//----------------------------------------------------------------------------//
//            Copyright 2018 Rieckermann Engineering Operations               //
//                Automatically Generated File - Do Not Edit                  //
//----------------------------------------------------------------------------//
// Description:                                                               //
// This file contains globally addressable event words for process alarms and //
// messages to be logged.                                                     //
//----------------------------------------------------------------------------//
// Revision history:                                                          //
// Rev By               Date        CC        Note                            //
// 1.1 David Paspa      10-Aug-2018 NA        Convert triggers to word bits.  //
// 1.0 David Paspa      14-May-2018 NA        Initial design for S7-1500.     //
//----------------------------------------------------------------------------//
DATA_BLOCK "dbEVENT"
TITLE = Global messages bits
{ S7_Optimized_Access := 'TRUE' }
AUTHOR : REO
NAME : dbEVENT
VERSION : 1.1

STRUCT
    alarmBlock : STRUCT                          // Block related alarms
@@TEMPLATE_BEGIN|createLevelsGlobal@@
@@ATTR_BEGIN|createClassesForLevel@@
@@ATTR_BEGIN|createInstancesGlobal@@
        alarm_@@INSTANCE@@ : Int;                // @@CLASS@@ block alarms
@@ATTR_END|createInstancesGlobal@@
@@ATTR_END|createClassesForLevel@@
@@TEMPLATE_END@@
    END_STRUCT ;
    eventConfirmNo : STRUCT                         // SFC events for logging prompt confirm No
@@TEMPLATE_BEGIN|INSTANCE_BLK_ALL@@
@@ATTR_BEGIN|pEventConfirmNoWordInstance@@
        event_@@INSTANCE@@_@@CWORD@@ : Int;
@@ATTR_END|pEventConfirmNoWordInstance@@
@@TEMPLATE_END@@
    END_STRUCT ;
    eventConfirmYes : STRUCT                             // SFC events for logging prompt confirm Yes
@@TEMPLATE_BEGIN|INSTANCE_BLK_ALL@@
@@ATTR_BEGIN|pEventConfirmYesWordInstance@@
        event_@@INSTANCE@@_@@CWORD@@ : Int;
@@ATTR_END|pEventConfirmYesWordInstance@@
@@TEMPLATE_END@@
    END_STRUCT ;
    eventLogMsg : STRUCT                         // SFC events for logging messages
@@TEMPLATE_BEGIN|INSTANCE_BLK_ALL@@
@@ATTR_BEGIN|pEventLogMsgWordInstance@@
        event_@@INSTANCE@@_@@CWORD@@ : Int;
@@ATTR_END|pEventLogMsgWordInstance@@
@@TEMPLATE_END@@
    END_STRUCT ;
    eventLogReal : STRUCT                        // SFC events for logging Real data
@@TEMPLATE_BEGIN|INSTANCE_BLK_ALL@@
@@ATTR_BEGIN|pEventLogRealWordInstance@@
        event_@@INSTANCE@@_@@CWORD@@ : Int;
@@ATTR_END|pEventLogRealWordInstance@@
@@TEMPLATE_END@@
    END_STRUCT ;
@@TEMPLATE_BEGIN|pEventLogTimeExists@@
    eventLogTime : STRUCT                        // SFC events for logging Time data
@@ATTR_BEGIN|INSTANCE_BLK_ALL@@
@@ATTR_BEGIN|pEventLogTimeWordInstance@@
        event_@@INSTANCE@@_@@CWORD@@ : Int;
@@ATTR_END|pEventLogTimeWordInstance@@
@@ATTR_END|INSTANCE_BLK_ALL@@
    END_STRUCT ;
@@TEMPLATE_END@@
@@TEMPLATE_BEGIN|pEventLogRealNumAll@@
    eventDataReal : Array[0..@@IDXEVENTMAX@@] of Real;   // SFC events for logging real data
@@TEMPLATE_END@@
@@TEMPLATE_BEGIN|pEventLogTimeExists@@
@@ATTR_BEGIN|pEventLogTimeNumAll@@
    eventDataTime : Array[0..@@IDXEVENTMAX@@] of DWord;  // SFC events for logging tmie data
@@ATTR_END|pEventLogTimeNumAll@@
@@TEMPLATE_END@@
    eventPrompt : STRUCT                         // SFC events for operator prompts
@@TEMPLATE_BEGIN|pEventPromptNum@@
        event : Array[1..@@IDXEVENTMAX@@] of "udtEventPrompt";
@@TEMPLATE_END@@
    END_STRUCT ;
END_STRUCT;

BEGIN
END_DATA_BLOCK
